// SIMATIC S7-200 project (STEP 7-Micro/WIN), CPU 222 REL 02.01

SYMBOL_TABLE USUARIO1
PARO             I0.0
MARCHA           I0.1
LAMPARA          Q0.0
END_SYMBOL_TABLE

ORGANIZATION_BLOCK PRINCIPAL:OB1
TITLE=COMENTARIOS DEL PROGRAMA
BEGIN
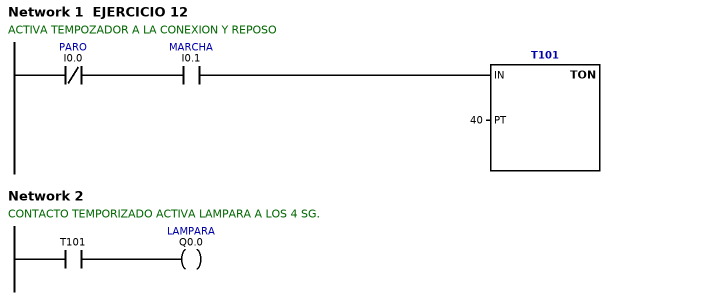
Network 1 // EJERCICIO 12
// ACTIVA TEMPOZADOR A LA CONEXION Y REPOSO
// (network saved uncompiled; LAD cells follow)
// row 0: c0 -|/|- PARO:I0.0  c1 -| |- MARCHA:I0.1  c2 --  c3 --  c4 [TON T101 IN:=power@row0, PT:=40]
// row 1: c4 [box]
Network 2
// CONTACTO TEMPORIZADO ACTIVA LAMPARA A LOS 4 SG.
// (network saved uncompiled; LAD cells follow)
// row 0: c0 -| |- T101  c1 -( ) LAMPARA:Q0.0
END_ORGANIZATION_BLOCK
